   t5[490] := 0.023831;
   t5[491] := 0.0266696;
   t5[492] := 0.0293428;
   t5[493] := 0.0318604;
   t5[494] := 0.0342322;
   t5[495] := -0.0208986;
   t5[496] := -0.0225395;
   t5[497] := -0.0240864;
   t5[498] := -0.0255261;
   t5[499] := -0.0268454;
   t5[500] := -0.0280312;
   t5[501] := -0.0290703;
   t5[502] := -0.0299495;
   t5[503] := -0.0306555;
   t5[504] := -0.0311752;
   t5[505] := -0.0314958;
   t5[506] := -0.0316138;
   t5[507] := -0.0315351;
   t5[508] := -0.0312663;
   t5[509] := -0.0308137;
   t5[510] := -0.0136591;
   t5[511] := -0.0122989;
   t5[512] := -0.0110547;
   t5[513] := -0.0099303;
   t5[514] := -0.0089297;
   t5[515] := -0.0080568;
   t5[516] := -0.0073155;
   t5[517] := -0.0067099;
   t5[518] := -0.0062437;
   t5[519] := -0.0059209;
   t5[520] := -0.0057453;
   t5[521] := -0.0057154;
   t5[522] := -0.0058246;
   t5[523] := -0.006066;
   t5[524] := -0.0064327;
   t5[525] := -0.014299;
   t5[526] := -0.0104196;
   t5[527] := -0.0064601;
   t5[528] := -0.0024202;
   t5[529] := 0.0017005;
   t5[530] := 0.0059023;
   t5[531] := 0.0101856;
   t5[532] := 0.0145506;
   t5[533] := 0.0189979;
   t5[534] := 0.0235277;
   t5[535] := 0.0281401;
   t5[536] := 0.0328307;
   t5[537] := 0.0375902;
   t5[538] := 0.042409;
   t5[539] := 0.0472775;
   t5[540] := -0.0809446;
   t5[541] := -0.0816613;
   t5[542] := -0.0823782;
   t5[543] := -0.0831006;
   t5[544] := -0.0838339;
   t5[545] := -0.0845833;
   t5[546] := -0.0853541;
   t5[547] := -0.0861518;
   t5[548] := -0.0869815;
   t5[549] := -0.0878487;
   t5[550] := -0.0887583;
   t5[551] := -0.0897094;
   t5[552] := -0.0906944;
   t5[553] := -0.0917059;
   t5[554] := -0.092736;
   t5[555] := 0.0001257;
   t5[556] := 0.0029497;
   t5[557] := 0.0057871;
   t5[558] := 0.0086392;
   t5[559] := 0.0115078;
   t5[560] := 0.0143943;
   t5[561] := 0.0173003;
   t5[562] := 0.0202273;
   t5[563] := 0.0231768;
   t5[564] := 0.0261505;
   t5[565] := 0.0291498;
   t5[566] := 0.0321767;
   t5[567] := 0.0352333;
   t5[568] := 0.0383218;
   t5[569] := 0.0414445;
   t5[570] := -0.0673197;
   t5[571] := -0.0670321;
   t5[572] := -0.0666434;
   t5[573] := -0.0661514;
   t5[574] := -0.0655542;
   t5[575] := -0.0648497;
   t5[576] := -0.0640358;
   t5[577] := -0.0631107;
   t5[578] := -0.0620721;
   t5[579] := -0.0609182;
   t5[580] := -0.0596471;
   t5[581] := -0.0582624;
   t5[582] := -0.0567733;
   t5[583] := -0.0551894;
   t5[584] := -0.05352;
   t5[585] := 0.0792828;
   t5[586] := 0.0762561;
   t5[587] := 0.073232;
   t5[588] := 0.0702186;
   t5[589] := 0.067224;
   t5[590] := 0.0642562;
   t5[591] := 0.0613231;
   t5[592] := 0.058433;
   t5[593] := 0.0555937;
   t5[594] := 0.0528132;
   t5[595] := 0.0500996;
   t5[596] := 0.0474569;
   t5[597] := 0.0448857;
   t5[598] := 0.042386;
   t5[599] := 0.0399582;
   t5[600] := -0.1993882;
   t5[601] := -0.1970195;
   t5[602] := -0.1945705;
   t5[603] := -0.1920432;
   t5[604] := -0.1894396;
   t5[605] := -0.1867614;
   t5[606] := -0.1840106;
   t5[607] := -0.1811892;
   t5[608] := -0.1782989;
   t5[609] := -0.1753418;
   t5[610] := -0.1723197;
   t5[611] := -0.1692367;
   t5[612] := -0.1660989;
   t5[613] := -0.1629122;
   t5[614] := -0.159683;
   t5[615] := -0.110986;
   t5[616] := -0.112907;
   t5[617] := -0.1145904;
   t5[618] := -0.11603;
   t5[619] := -0.1172196;
   t5[620] := -0.118153;
   t5[621] := -0.1188239;
   t5[622] := -0.119226;
   t5[623] := -0.1193531;
   t5[624] := -0.1191991;
   t5[625] := -0.1187581;
   t5[626] := -0.1180348;
   t5[627] := -0.1170453;
   t5[628] := -0.1158056;
   t5[629] := -0.1143322;
   t5[630] := -0.0163093;
   t5[631] := -0.0198292;
   t5[632] := -0.0232166;
   t5[633] := -0.0264609;
   t5[634] := -0.0295518;
   t5[635] := -0.0324788;
   t5[636] := -0.0352314;
   t5[637] := -0.0377992;
   t5[638] := -0.0401717;
   t5[639] := -0.0423386;
   t5[640] := -0.0442896;
   t5[641] := -0.0460239;
   t5[642] := -0.0475501;
   t5[643] := -0.0488771;
   t5[644] := -0.0500139;
   t5[645] := 0.0848828;
   t5[646] := 0.0819437;
   t5[647] := 0.0790844;
   t5[648] := 0.0763136;
   t5[649] := 0.0736399;
   t5[650] := 0.0710721;
   t5[651] := 0.0686188;
   t5[652] := 0.0662886;
   t5[653] := 0.0640904;
   t5[654] := 0.0620326;
   t5[655] := 0.0601237;
   t5[656] := 0.0583629;
   t5[657] := 0.05674;
   t5[658] := 0.0552444;
   t5[659] := 0.0538658;
   t5[660] := -0.0819279;
   t5[661] := -0.0837696;
   t5[662] := -0.085415;
   t5[663] := -0.0868444;
   t5[664] := -0.088038;
   t5[665] := -0.0889764;
   t5[666] := -0.0896396;
   t5[667] := -0.0900081;
   t5[668] := -0.0900622;
   t5[669] := -0.0897822;
   t5[670] := -0.0891493;
   t5[671] := -0.0881638;
   t5[672] := -0.0868462;
   t5[673] := -0.0852177;
   t5[674] := -0.0832996;
   t5[675] := -0.0222091;
   t5[676] := -0.019204;
   t5[677] := -0.0163363;
   t5[678] := -0.0136269;
   t5[679] := -0.0110964;
   t5[680] := -0.0087656;
   t5[681] := -0.0066552;
   t5[682] := -0.004786;
   t5[683] := -0.0031786;
   t5[684] := -0.0018538;
   t5[685] := -0.0008317;
   t5[686] := -0.0001178;
   t5[687] := 0.0002977;
   t5[688] := 0.0004254;
   t5[689] := 0.0002755;
   t5[690] := -0.0469918;
   t5[691] := -0.0436484;
   t5[692] := -0.0405246;
   t5[693] := -0.0376308;
   t5[694] := -0.0349775;
   t5[695] := -0.0325752;
   t5[696] := -0.0304344;
   t5[697] := -0.0285657;
   t5[698] := -0.0269795;
   t5[699] := -0.0256863;
   t5[700] := -0.0246962;
   t5[701] := -0.0240066;
   t5[702] := -0.0236022;
   t5[703] := -0.0234672;
   t5[704] := -0.0235855;
   t5[705] := 0.0315658;
   t5[706] := 0.0328791;
   t5[707] := 0.0340612;
   t5[708] := 0.0351116;
   t5[709] := 0.0360298;
   t5[710] := 0.0368152;
   t5[711] := 0.0374672;
   t5[712] := 0.0379854;
   t5[713] := 0.0383692;
   t5[714] := 0.038618;
   t5[715] := 0.0387315;
   t5[716] := 0.0387144;
   t5[717] := 0.0385764;
   t5[718] := 0.0383273;
   t5[719] := 0.0379772;
   t5[720] := 0.0589575;
   t5[721] := 0.0571638;
   t5[722] := 0.0552337;
   t5[723] := 0.0531697;
   t5[724] := 0.0509741;
   t5[725] := 0.0486495;
   t5[726] := 0.0461984;
   t5[727] := 0.0436231;
   t5[728] := 0.0409261;
   t5[729] := 0.03811;
   t5[730] := 0.0351772;
   t5[731] := 0.0321336;
   t5[732] := 0.0289883;
   t5[733] := 0.0257505;
   t5[734] := 0.0224294;
   t5[735] := -0.0370074;
   t5[736] := -0.0344528;
   t5[737] := -0.0317711;
   t5[738] := -0.0289586;
   t5[739] := -0.0260112;
   t5[740] := -0.022925;
   t5[741] := -0.0196963;
   t5[742] := -0.016321;
   t5[743] := -0.0127952;
   t5[744] := -0.0091151;
   t5[745] := -0.005277;
   t5[746] := -0.0012858;
   t5[747] := 0.0028455;
   t5[748] := 0.007103;
   t5[749] := 0.0114734;
   t5[750] := -0.0503424;
   t5[751] := -0.0554995;
   t5[752] := -0.0605443;
   t5[753] := -0.0654624;
   t5[754] := -0.0702395;
   t5[755] := -0.0748614;
   t5[756] := -0.0793139;
   t5[757] := -0.0835825;
   t5[758] := -0.087653;
   t5[759] := -0.0915111;
   t5[760] := -0.095143;
   t5[761] := -0.0985424;
   t5[762] := -0.1017114;
   t5[763] := -0.1046524;
   t5[764] := -0.1073677;
   t5[765] := -0.1648159;
   t5[766] := -0.1596806;
   t5[767] := -0.1543417;
   t5[768] := -0.1488126;
   t5[769] := -0.1431066;
   t5[770] := -0.1372371;
   t5[771] := -0.1312175;
   t5[772] := -0.1250611;
   t5[773] := -0.1187812;
   t5[774] := -0.1123913;
   t5[775] := -0.1059046;
   t5[776] := -0.0993333;
   t5[777] := -0.0926887;
   t5[778] := -0.0859816;
   t5[779] := -0.0792232;
   t5[780] := -0.0904827;
   t5[781] := -0.0898896;
   t5[782] := -0.0893127;
   t5[783] := -0.0887551;
   t5[784] := -0.0882202;
   t5[785] := -0.0877112;
   t5[786] := -0.0872314;
   t5[787] := -0.0867841;
   t5[788] := -0.0863725;
   t5[789] := -0.0859999;
   t5[790] := -0.0856695;
   t5[791] := -0.0853802;
   t5[792] := -0.0851272;
   t5[793] := -0.0849053;
   t5[794] := -0.0847093;
   t5[795] := -0.0673839;
   t5[796] := -0.0627446;
   t5[797] := -0.0580462;
   t5[798] := -0.0533;
   t5[799] := -0.0485171;
   t5[800] := -0.0437086;
   t5[801] := -0.0388857;
   t5[802] := -0.0340594;
   t5[803] := -0.0292411;
   t5[804] := -0.0244417;
   t5[805] := -0.0196723;
   t5[806] := -0.0149416;
   t5[807] := -0.0102555;
   t5[808] := -0.0056201;
   t5[809] := -0.0010412;
   t5[810] := 0.075334;
   t5[811] := 0.0749833;
   t5[812] := 0.0743661;
   t5[813] := 0.0734706;
   t5[814] := 0.072285;
   t5[815] := 0.0707974;
   t5[816] := 0.068996;
   t5[817] := 0.0668689;
   t5[818] := 0.0644045;
   t5[819] := 0.0615908;
   t5[820] := 0.0584166;
   t5[821] := 0.0548866;
   t5[822] := 0.0510212;
   t5[823] := 0.0468419;
   t5[824] := 0.04237;
   t5[825] := -0.1063465;
   t5[826] := -0.1045535;
   t5[827] := -0.1026798;
   t5[828] := -0.1007291;
   t5[829] := -0.0987055;
   t5[830] := -0.0966127;
   t5[831] := -0.0944546;
   t5[832] := -0.092235;
   t5[833] := -0.0899577;
   t5[834] := -0.0876267;
   t5[835] := -0.0852457;
   t5[836] := -0.0828167;
   t5[837] := -0.0803401;
   t5[838] := -0.077816;
   t5[839] := -0.0752449;
   t5[840] := 0.0025241;
   t5[841] := 0.0003729;
   t5[842] := -0.0018117;
   t5[843] := -0.0040243;
   t5[844] := -0.0062591;
   t5[845] := -0.0085107;
   t5[846] := -0.0107734;
   t5[847] := -0.0130416;
   t5[848] := -0.0153097;
   t5[849] := -0.0175722;
   t5[850] := -0.0198235;
   t5[851] := -0.0220606;
   t5[852] := -0.0242824;
   t5[853] := -0.0264882;
   t5[854] := -0.0286772;
   t5[855] := -0.0587365;
   t5[856] := -0.0658987;
   t5[857] := -0.0729648;
   t5[858] := -0.07991;
   t5[859] := -0.0867094;
   t5[860] := -0.0933378;
   t5[861] := -0.0997704;
   t5[862] := -0.1059823;
   t5[863] := -0.1119484;
   t5[864] := -0.1176438;
   t5[865] := -0.1230443;
   t5[866] := -0.1281403;
   t5[867] := -0.1329374;
   t5[868] := -0.137442;
   t5[869] := -0.1416606;
   t5[870] := -0.0241061;
   t5[871] := -0.0227329;
   t5[872] := -0.0212774;
   t5[873] := -0.0197337;
   t5[874] := -0.0180954;
   t5[875] := -0.0163565;
   t5[876] := -0.0145109;
   t5[877] := -0.0125525;
   t5[878] := -0.0104751;
   t5[879] := -0.0082726;
   t5[880] := -0.0059392;
   t5[881] := -0.0034767;
   t5[882] := -0.0008946;
   t5[883] := 0.001797;
   t5[884] := 0.0045883;
   t5[885] := -0.016338;
   t5[886] := -0.0135221;
   t5[887] := -0.0107115;
   t5[888] := -0.0079037;
   t5[889] := -0.0050963;
   t5[890] := -0.0022869;
   t5[891] := 0.0005271;
   t5[892] := 0.0033482;
   t5[893] := 0.0061787;
   t5[894] := 0.0090212;
   t5[895] := 0.011878;
   t5[896] := 0.0147486;
   t5[897] := 0.0176293;
   t5[898] := 0.0205164;
   t5[899] := 0.0234063;
   t5[900] := -0.0519279;
   t5[901] := -0.056473;
   t5[902] := -0.0609004;
   t5[903] := -0.0652012;
   t5[904] := -0.0693667;
   t5[905] := -0.0733882;
   t5[906] := -0.0772569;
   t5[907] := -0.0809641;
   t5[908] := -0.0845011;
   t5[909] := -0.087859;
   t5[910] := -0.0910294;
   t5[911] := -0.0940104;
   t5[912] := -0.0968068;
   t5[913] := -0.0994238;
   t5[914] := -0.1018665;
   t5[915] := 0.142846;
   t5[916] := 0.1405271;
   t5[917] := 0.1380653;
   t5[918] := 0.1354591;
   t5[919] := 0.1327065;
   t5[920] := 0.129806;
   t5[921] := 0.1267559;
   t5[922] := 0.1235543;
   t5[923] := 0.1201996;
   t5[924] := 0.11669;
   t5[925] := 0.1130242;
   t5[926] := 0.109206;
   t5[927] := 0.1052453;
   t5[928] := 0.1011521;
   t5[929] := 0.0969364;
   t5[930] := -0.0299947;
   t5[931] := -0.0294521;
   t5[932] := -0.0288785;
   t5[933] := -0.0282723;
   t5[934] := -0.0276319;
   t5[935] := -0.0269553;
   t5[936] := -0.0262411;
   t5[937] := -0.0254874;
   t5[938] := -0.0246926;
   t5[939] := -0.0238549;
   t5[940] := -0.0229728;
   t5[941] := -0.0220476;
   t5[942] := -0.0210837;
   t5[943] := -0.0200855;
   t5[944] := -0.0190576;
   t5[945] := -0.0100999;
   t5[946] := -0.0030712;
   t5[947] := 0.0037406;
   t5[948] := 0.0103103;
   t5[949] := 0.0166126;
   t5[950] := 0.0226221;
   t5[951] := 0.0283136;
   t5[952] := 0.0336617;
   t5[953] := 0.038641;
   t5[954] := 0.0432264;
   t5[955] := 0.0473932;
   t5[956] := 0.0511381;
   t5[957] := 0.054479;
   t5[958] := 0.0574348;
   t5[959] := 0.0600244;
   w6[0] := 0.0254122;
   w6[1] := -0.4251655;
   w6[2] := -0.4513899;
   w6[3] := 0.0262705;
   w6[4] := 0.3702881;
   w6[5] := -0.1208161;
   w6[6] := -0.2231239;
   w6[7] := 0.2512441;
   w6[8] := -0.3278799;
   w6[9] := 0.2889541;
   w6[10] := -0.0654242;
   w6[11] := 0.1067281;
   w6[12] := 0.2623815;
   w6[13] := -0.1798091;
   w6[14] := -0.3070911;
   w6[15] := -0.4204447;
   w6[16] := 0.5762351;
   w6[17] := -1.090657;
   w6[18] := -0.2690518;
   w6[19] := -0.6730261;
   w6[20] := -0.0514923;
   w6[21] := -0.4457789;
   w6[22] := 0.5072183;
   w6[23] := -0.0549661;
   w6[24] := 0.3812394;
   w6[25] := -0.606307;
   w6[26] := 0.1917919;
   w6[27] := 0.1525442;
   w6[28] := -0.4219312;
   w6[29] := 0.338313;
   w6[30] := 0.1919874;
   w6[31] := -0.3457294;
   w6[32] := 0.1728978;
   w6[33] := 0.5825878;
   w6[34] := 0.7331663;
   w6[35] := 0.4268312;
   w6[36] := -0.0077422;
   w6[37] := 0.4766487;
   w6[38] := 0.102607;
   w6[39] := -0.5723706;
   w6[40] := 0.0728498;
   w6[41] := 0.4253429;
   w6[42] := -0.3637053;
   w6[43] := -0.6206156;
   w6[44] := 0.2656944;
   w6[45] := -0.3130539;
   w6[46] := 0.2033212;
   w6[47] := 0.1327122;
   w6[48] := -0.709101;
   w6[49] := 0.7231103;
   w6[50] := -0.2214241;
   w6[51] := 0.4491622;
   w6[52] := -0.3655713;
   w6[53] := 0.4263724;
   w6[54] := 0.0266531;
   w6[55] := 0.4637966;
   w6[56] := -0.3418979;
   w6[57] := -0.2391363;
   w6[58] := 0.4152579;
   w6[59] := 0.2146362;
   w6[60] := -0.3901598;
   w6[61] := -0.1938754;
   w6[62] := -0.561949;
   w6[63] := 0.4047181;
END_DATA_BLOCK

FUNCTION_BLOCK "NeuroPLC_Inference"   // FB1, SCL
{ S7_Optimized_Access := 'FALSE' }
VERSION : 0.1
// NeuroPLC 鈥?Auto-generated IEC 61131-3 SCL (DB+FB Mode)
//  Graph: kan | Target: S71200DBBackend
//  Work memory: 75KB | LUT points: 15
//  Nodes: 11 | Ops: {'matmul': 3, 'standard_act': 2, 'bspline_lut': 2, 'add': 2, 'softmax': 1, 'argmax': 1}
//  Parameters in DB "NeuroPLC_KAN_Weights", inference in FB.
   VAR_INPUT
      features : Array[0..27] of Real;   // 28-D feature vector
   END_VAR
   VAR_OUTPUT
      fault_class : Int;   // 0=Normal, 1=InnerRace, 2=Ball, 3=OuterRace
      confidence : Real;   // max softmax probability 鈹€鈹€ Inference temporaries 鈹€鈹€
   END_VAR
   VAR
      v1 : Array[0..27] of Real;   // silu output
      v3 : Array[0..447] of Real;   // BsplineLUT output (1D: o*28+i)
      v2 : Array[0..15] of Real;   // matmul output
      v4 : Array[0..15] of Real;   // add merge
      v5 : Array[0..15] of Real;   // silu output
      v7 : Array[0..63] of Real;   // BsplineLUT output (1D: o*16+i)
      v6 : Array[0..3] of Real;   // matmul output
      v8 : Array[0..3] of Real;   // add merge
      v9 : Array[0..3] of Real;   // softmax output 鈹€鈹€ Temporary variables 鈹€鈹€
      i : Int;
      o : Int;
      j : Int;
      lo : Int;
      hi : Int;
      idx : Int;
      base : Int;
      sum : Real;
      max_val : Real;
      t_val : Real;
   END_VAR
BEGIN
      // 鈺愨晲鈺?Inference forward pass 鈺愨晲鈺?
       // Parameters loaded from DB "NeuroPLC_KAN_Weights" (start values = data, not code)

          // Input: features[0..27]

          // StandardAct: silu
          FOR #i := 0 TO 27 DO
              // SiLU = x / (1 + exp(-x))
              #v1[#i] := #features[#i] / (1.0 + EXP(-#features[#i]));
          END_FOR;

          // BsplineLUT: l0_bspline (16x28, 15 pts)
          FOR #i := 0 TO 27 DO
              // Linear scan: find largest grid[j] <= input[i]
              #lo := 0;
              FOR #j := 1 TO 13 DO
                  IF #features[#i] >= "NeuroPLC_KAN_Weights".g0[#j] THEN
                      #lo := #j;
                  END_IF;
              END_FOR;
              #hi := #lo + 1;
              #t_val := (#features[#i] - "NeuroPLC_KAN_Weights".g0[#lo]) /
                        ("NeuroPLC_KAN_Weights".g0[#hi] - "NeuroPLC_KAN_Weights".g0[#lo] + 1.0E-10);
              FOR #o := 0 TO 15 DO
                  #base := (#o * 28 + #i) * 15;
                  #idx := #o * 28 + #i;
                  #v3[#idx] :=
                      "NeuroPLC_KAN_Weights".t1[#base + #lo] * (1.0 - #t_val) +
                      "NeuroPLC_KAN_Weights".t1[#base + #hi] * #t_val;
              END_FOR;
          END_FOR;

          // MatMul: l0_base
          #v2[0] := "NeuroPLC_KAN_Weights".b3[0] + "NeuroPLC_KAN_Weights".w2[0] * #v1[0] + "NeuroPLC_KAN_Weights".w2[1] * #v1[1] + "NeuroPLC_KAN_Weights".w2[2] * #v1[2] + "NeuroPLC_KAN_Weights".w2[3] * #v1[3] + "NeuroPLC_KAN_Weights".w2[4] * #v1[4] + "NeuroPLC_KAN_Weights".w2[5] * #v1[5] + "NeuroPLC_KAN_Weights".w2[6] * #v1[6] + "NeuroPLC_KAN_Weights".w2[7] * #v1[7] + "NeuroPLC_KAN_Weights".w2[8] * #v1[8] + "NeuroPLC_KAN_Weights".w2[9] * #v1[9] + "NeuroPLC_KAN_Weights".w2[10] * #v1[10] + "NeuroPLC_KAN_Weights".w2[11] * #v1[11] + "NeuroPLC_KAN_Weights".w2[12] * #v1[12] + "NeuroPLC_KAN_Weights".w2[13] * #v1[13] + "NeuroPLC_KAN_Weights".w2[14] * #v1[14] + "NeuroPLC_KAN_Weights".w2[15] * #v1[15] + "NeuroPLC_KAN_Weights".w2[16] * #v1[16] + "NeuroPLC_KAN_Weights".w2[17] * #v1[17] + "NeuroPLC_KAN_Weights".w2[18] * #v1[18] + "NeuroPLC_KAN_Weights".w2[19] * #v1[19] + "NeuroPLC_KAN_Weights".w2[20] * #v1[20] + "NeuroPLC_KAN_Weights".w2[21] * #v1[21] + "NeuroPLC_KAN_Weights".w2[22] * #v1[22] + "NeuroPLC_KAN_Weights".w2[23] * #v1[23] + "NeuroPLC_KAN_Weights".w2[24] * #v1[24] + "NeuroPLC_KAN_Weights".w2[25] * #v1[25] + "NeuroPLC_KAN_Weights".w2[26] * #v1[26] + "NeuroPLC_KAN_Weights".w2[27] * #v1[27];
          #v2[1] := "NeuroPLC_KAN_Weights".b3[1] + "NeuroPLC_KAN_Weights".w2[28] * #v1[0] + "NeuroPLC_KAN_Weights".w2[29] * #v1[1] + "NeuroPLC_KAN_Weights".w2[30] * #v1[2] + "NeuroPLC_KAN_Weights".w2[31] * #v1[3] + "NeuroPLC_KAN_Weights".w2[32] * #v1[4] + "NeuroPLC_KAN_Weights".w2[33] * #v1[5] + "NeuroPLC_KAN_Weights".w2[34] * #v1[6] + "NeuroPLC_KAN_Weights".w2[35] * #v1[7] + "NeuroPLC_KAN_Weights".w2[36] * #v1[8] + "NeuroPLC_KAN_Weights".w2[37] * #v1[9] + "NeuroPLC_KAN_Weights".w2[38] * #v1[10] + "NeuroPLC_KAN_Weights".w2[39] * #v1[11] + "NeuroPLC_KAN_Weights".w2[40] * #v1[12] + "NeuroPLC_KAN_Weights".w2[41] * #v1[13] + "NeuroPLC_KAN_Weights".w2[42] * #v1[14] + "NeuroPLC_KAN_Weights".w2[43] * #v1[15] + "NeuroPLC_KAN_Weights".w2[44] * #v1[16] + "NeuroPLC_KAN_Weights".w2[45] * #v1[17] + "NeuroPLC_KAN_Weights".w2[46] * #v1[18] + "NeuroPLC_KAN_Weights".w2[47] * #v1[19] + "NeuroPLC_KAN_Weights".w2[48] * #v1[20] + "NeuroPLC_KAN_Weights".w2[49] * #v1[21] + "NeuroPLC_KAN_Weights".w2[50] * #v1[22] + "NeuroPLC_KAN_Weights".w2[51] * #v1[23] + "NeuroPLC_KAN_Weights".w2[52] * #v1[24] + "NeuroPLC_KAN_Weights".w2[53] * #v1[25] + "NeuroPLC_KAN_Weights".w2[54] * #v1[26] + "NeuroPLC_KAN_Weights".w2[55] * #v1[27];
          #v2[2] := "NeuroPLC_KAN_Weights".b3[2] + "NeuroPLC_KAN_Weights".w2[56] * #v1[0] + "NeuroPLC_KAN_Weights".w2[57] * #v1[1] + "NeuroPLC_KAN_Weights".w2[58] * #v1[2] + "NeuroPLC_KAN_Weights".w2[59] * #v1[3] + "NeuroPLC_KAN_Weights".w2[60] * #v1[4] + "NeuroPLC_KAN_Weights".w2[61] * #v1[5] + "NeuroPLC_KAN_Weights".w2[62] * #v1[6] + "NeuroPLC_KAN_Weights".w2[63] * #v1[7] + "NeuroPLC_KAN_Weights".w2[64] * #v1[8] + "NeuroPLC_KAN_Weights".w2[65] * #v1[9] + "NeuroPLC_KAN_Weights".w2[66] * #v1[10] + "NeuroPLC_KAN_Weights".w2[67] * #v1[11] + "NeuroPLC_KAN_Weights".w2[68] * #v1[12] + "NeuroPLC_KAN_Weights".w2[69] * #v1[13] + "NeuroPLC_KAN_Weights".w2[70] * #v1[14] + "NeuroPLC_KAN_Weights".w2[71] * #v1[15] + "NeuroPLC_KAN_Weights".w2[72] * #v1[16] + "NeuroPLC_KAN_Weights".w2[73] * #v1[17] + "NeuroPLC_KAN_Weights".w2[74] * #v1[18] + "NeuroPLC_KAN_Weights".w2[75] * #v1[19] + "NeuroPLC_KAN_Weights".w2[76] * #v1[20] + "NeuroPLC_KAN_Weights".w2[77] * #v1[21] + "NeuroPLC_KAN_Weights".w2[78] * #v1[22] + "NeuroPLC_KAN_Weights".w2[79] * #v1[23] + "NeuroPLC_KAN_Weights".w2[80] * #v1[24] + "NeuroPLC_KAN_Weights".w2[81] * #v1[25] + "NeuroPLC_KAN_Weights".w2[82] * #v1[26] + "NeuroPLC_KAN_Weights".w2[83] * #v1[27];
          #v2[3] := "NeuroPLC_KAN_Weights".b3[3] + "NeuroPLC_KAN_Weights".w2[84] * #v1[0] + "NeuroPLC_KAN_Weights".w2[85] * #v1[1] + "NeuroPLC_KAN_Weights".w2[86] * #v1[2] + "NeuroPLC_KAN_Weights".w2[87] * #v1[3] + "NeuroPLC_KAN_Weights".w2[88] * #v1[4] + "NeuroPLC_KAN_Weights".w2[89] * #v1[5] + "NeuroPLC_KAN_Weights".w2[90] * #v1[6] + "NeuroPLC_KAN_Weights".w2[91] * #v1[7] + "NeuroPLC_KAN_Weights".w2[92] * #v1[8] + "NeuroPLC_KAN_Weights".w2[93] * #v1[9] + "NeuroPLC_KAN_Weights".w2[94] * #v1[10] + "NeuroPLC_KAN_Weights".w2[95] * #v1[11] + "NeuroPLC_KAN_Weights".w2[96] * #v1[12] + "NeuroPLC_KAN_Weights".w2[97] * #v1[13] + "NeuroPLC_KAN_Weights".w2[98] * #v1[14] + "NeuroPLC_KAN_Weights".w2[99] * #v1[15] + "NeuroPLC_KAN_Weights".w2[100] * #v1[16] + "NeuroPLC_KAN_Weights".w2[101] * #v1[17] + "NeuroPLC_KAN_Weights".w2[102] * #v1[18] + "NeuroPLC_KAN_Weights".w2[103] * #v1[19] + "NeuroPLC_KAN_Weights".w2[104] * #v1[20] + "NeuroPLC_KAN_Weights".w2[105] * #v1[21] + "NeuroPLC_KAN_Weights".w2[106] * #v1[22] + "NeuroPLC_KAN_Weights".w2[107] * #v1[23] + "NeuroPLC_KAN_Weights".w2[108] * #v1[24] + "NeuroPLC_KAN_Weights".w2[109] * #v1[25] + "NeuroPLC_KAN_Weights".w2[110] * #v1[26] + "NeuroPLC_KAN_Weights".w2[111] * #v1[27];
          #v2[4] := "NeuroPLC_KAN_Weights".b3[4] + "NeuroPLC_KAN_Weights".w2[112] * #v1[0] + "NeuroPLC_KAN_Weights".w2[113] * #v1[1] + "NeuroPLC_KAN_Weights".w2[114] * #v1[2] + "NeuroPLC_KAN_Weights".w2[115] * #v1[3] + "NeuroPLC_KAN_Weights".w2[116] * #v1[4] + "NeuroPLC_KAN_Weights".w2[117] * #v1[5] + "NeuroPLC_KAN_Weights".w2[118] * #v1[6] + "NeuroPLC_KAN_Weights".w2[119] * #v1[7] + "NeuroPLC_KAN_Weights".w2[120] * #v1[8] + "NeuroPLC_KAN_Weights".w2[121] * #v1[9] + "NeuroPLC_KAN_Weights".w2[122] * #v1[10] + "NeuroPLC_KAN_Weights".w2[123] * #v1[11] + "NeuroPLC_KAN_Weights".w2[124] * #v1[12] + "NeuroPLC_KAN_Weights".w2[125] * #v1[13] + "NeuroPLC_KAN_Weights".w2[126] * #v1[14] + "NeuroPLC_KAN_Weights".w2[127] * #v1[15] + "NeuroPLC_KAN_Weights".w2[128] * #v1[16] + "NeuroPLC_KAN_Weights".w2[129] * #v1[17] + "NeuroPLC_KAN_Weights".w2[130] * #v1[18] + "NeuroPLC_KAN_Weights".w2[131] * #v1[19] + "NeuroPLC_KAN_Weights".w2[132] * #v1[20] + "NeuroPLC_KAN_Weights".w2[133] * #v1[21] + "NeuroPLC_KAN_Weights".w2[134] * #v1[22] + "NeuroPLC_KAN_Weights".w2[135] * #v1[23] + "NeuroPLC_KAN_Weights".w2[136] * #v1[24] + "NeuroPLC_KAN_Weights".w2[137] * #v1[25] + "NeuroPLC_KAN_Weights".w2[138] * #v1[26] + "NeuroPLC_KAN_Weights".w2[139] * #v1[27];
          #v2[5] := "NeuroPLC_KAN_Weights".b3[5] + "NeuroPLC_KAN_Weights".w2[140] * #v1[0] + "NeuroPLC_KAN_Weights".w2[141] * #v1[1] + "NeuroPLC_KAN_Weights".w2[142] * #v1[2] + "NeuroPLC_KAN_Weights".w2[143] * #v1[3] + "NeuroPLC_KAN_Weights".w2[144] * #v1[4] + "NeuroPLC_KAN_Weights".w2[145] * #v1[5] + "NeuroPLC_KAN_Weights".w2[146] * #v1[6] + "NeuroPLC_KAN_Weights".w2[147] * #v1[7] + "NeuroPLC_KAN_Weights".w2[148] * #v1[8] + "NeuroPLC_KAN_Weights".w2[149] * #v1[9] + "NeuroPLC_KAN_Weights".w2[150] * #v1[10] + "NeuroPLC_KAN_Weights".w2[151] * #v1[11] + "NeuroPLC_KAN_Weights".w2[152] * #v1[12] + "NeuroPLC_KAN_Weights".w2[153] * #v1[13] + "NeuroPLC_KAN_Weights".w2[154] * #v1[14] + "NeuroPLC_KAN_Weights".w2[155] * #v1[15] + "NeuroPLC_KAN_Weights".w2[156] * #v1[16] + "NeuroPLC_KAN_Weights".w2[157] * #v1[17] + "NeuroPLC_KAN_Weights".w2[158] * #v1[18] + "NeuroPLC_KAN_Weights".w2[159] * #v1[19] + "NeuroPLC_KAN_Weights".w2[160] * #v1[20] + "NeuroPLC_KAN_Weights".w2[161] * #v1[21] + "NeuroPLC_KAN_Weights".w2[162] * #v1[22] + "NeuroPLC_KAN_Weights".w2[163] * #v1[23] + "NeuroPLC_KAN_Weights".w2[164] * #v1[24] + "NeuroPLC_KAN_Weights".w2[165] * #v1[25] + "NeuroPLC_KAN_Weights".w2[166] * #v1[26] + "NeuroPLC_KAN_Weights".w2[167] * #v1[27];
          #v2[6] := "NeuroPLC_KAN_Weights".b3[6] + "NeuroPLC_KAN_Weights".w2[168] * #v1[0] + "NeuroPLC_KAN_Weights".w2[169] * #v1[1] + "NeuroPLC_KAN_Weights".w2[170] * #v1[2] + "NeuroPLC_KAN_Weights".w2[171] * #v1[3] + "NeuroPLC_KAN_Weights".w2[172] * #v1[4] + "NeuroPLC_KAN_Weights".w2[173] * #v1[5] + "NeuroPLC_KAN_Weights".w2[174] * #v1[6] + "NeuroPLC_KAN_Weights".w2[175] * #v1[7] + "NeuroPLC_KAN_Weights".w2[176] * #v1[8] + "NeuroPLC_KAN_Weights".w2[177] * #v1[9] + "NeuroPLC_KAN_Weights".w2[178] * #v1[10] + "NeuroPLC_KAN_Weights".w2[179] * #v1[11] + "NeuroPLC_KAN_Weights".w2[180] * #v1[12] + "NeuroPLC_KAN_Weights".w2[181] * #v1[13] + "NeuroPLC_KAN_Weights".w2[182] * #v1[14] + "NeuroPLC_KAN_Weights".w2[183] * #v1[15] + "NeuroPLC_KAN_Weights".w2[184] * #v1[16] + "NeuroPLC_KAN_Weights".w2[185] * #v1[17] + "NeuroPLC_KAN_Weights".w2[186] * #v1[18] + "NeuroPLC_KAN_Weights".w2[187] * #v1[19] + "NeuroPLC_KAN_Weights".w2[188] * #v1[20] + "NeuroPLC_KAN_Weights".w2[189] * #v1[21] + "NeuroPLC_KAN_Weights".w2[190] * #v1[22] + "NeuroPLC_KAN_Weights".w2[191] * #v1[23] + "NeuroPLC_KAN_Weights".w2[192] * #v1[24] + "NeuroPLC_KAN_Weights".w2[193] * #v1[25] + "NeuroPLC_KAN_Weights".w2[194] * #v1[26] + "NeuroPLC_KAN_Weights".w2[195] * #v1[27];
          #v2[7] := "NeuroPLC_KAN_Weights".b3[7] + "NeuroPLC_KAN_Weights".w2[196] * #v1[0] + "NeuroPLC_KAN_Weights".w2[197] * #v1[1] + "NeuroPLC_KAN_Weights".w2[198] * #v1[2] + "NeuroPLC_KAN_Weights".w2[199] * #v1[3] + "NeuroPLC_KAN_Weights".w2[200] * #v1[4] + "NeuroPLC_KAN_Weights".w2[201] * #v1[5] + "NeuroPLC_KAN_Weights".w2[202] * #v1[6] + "NeuroPLC_KAN_Weights".w2[203] * #v1[7] + "NeuroPLC_KAN_Weights".w2[204] * #v1[8] + "NeuroPLC_KAN_Weights".w2[205] * #v1[9] + "NeuroPLC_KAN_Weights".w2[206] * #v1[10] + "NeuroPLC_KAN_Weights".w2[207] * #v1[11] + "NeuroPLC_KAN_Weights".w2[208] * #v1[12] + "NeuroPLC_KAN_Weights".w2[209] * #v1[13] + "NeuroPLC_KAN_Weights".w2[210] * #v1[14] + "NeuroPLC_KAN_Weights".w2[211] * #v1[15] + "NeuroPLC_KAN_Weights".w2[212] * #v1[16] + "NeuroPLC_KAN_Weights".w2[213] * #v1[17] + "NeuroPLC_KAN_Weights".w2[214] * #v1[18] + "NeuroPLC_KAN_Weights".w2[215] * #v1[19] + "NeuroPLC_KAN_Weights".w2[216] * #v1[20] + "NeuroPLC_KAN_Weights".w2[217] * #v1[21] + "NeuroPLC_KAN_Weights".w2[218] * #v1[22] + "NeuroPLC_KAN_Weights".w2[219] * #v1[23] + "NeuroPLC_KAN_Weights".w2[220] * #v1[24] + "NeuroPLC_KAN_Weights".w2[221] * #v1[25] + "NeuroPLC_KAN_Weights".w2[222] * #v1[26] + "NeuroPLC_KAN_Weights".w2[223] * #v1[27];
          #v2[8] := "NeuroPLC_KAN_Weights".b3[8] + "NeuroPLC_KAN_Weights".w2[224] * #v1[0] + "NeuroPLC_KAN_Weights".w2[225] * #v1[1] + "NeuroPLC_KAN_Weights".w2[226] * #v1[2] + "NeuroPLC_KAN_Weights".w2[227] * #v1[3] + "NeuroPLC_KAN_Weights".w2[228] * #v1[4] + "NeuroPLC_KAN_Weights".w2[229] * #v1[5] + "NeuroPLC_KAN_Weights".w2[230] * #v1[6] + "NeuroPLC_KAN_Weights".w2[231] * #v1[7] + "NeuroPLC_KAN_Weights".w2[232] * #v1[8] + "NeuroPLC_KAN_Weights".w2[233] * #v1[9] + "NeuroPLC_KAN_Weights".w2[234] * #v1[10] + "NeuroPLC_KAN_Weights".w2[235] * #v1[11] + "NeuroPLC_KAN_Weights".w2[236] * #v1[12] + "NeuroPLC_KAN_Weights".w2[237] * #v1[13] + "NeuroPLC_KAN_Weights".w2[238] * #v1[14] + "NeuroPLC_KAN_Weights".w2[239] * #v1[15] + "NeuroPLC_KAN_Weights".w2[240] * #v1[16] + "NeuroPLC_KAN_Weights".w2[241] * #v1[17] + "NeuroPLC_KAN_Weights".w2[242] * #v1[18] + "NeuroPLC_KAN_Weights".w2[243] * #v1[19] + "NeuroPLC_KAN_Weights".w2[244] * #v1[20] + "NeuroPLC_KAN_Weights".w2[245] * #v1[21] + "NeuroPLC_KAN_Weights".w2[246] * #v1[22] + "NeuroPLC_KAN_Weights".w2[247] * #v1[23] + "NeuroPLC_KAN_Weights".w2[248] * #v1[24] + "NeuroPLC_KAN_Weights".w2[249] * #v1[25] + "NeuroPLC_KAN_Weights".w2[250] * #v1[26] + "NeuroPLC_KAN_Weights".w2[251] * #v1[27];
          #v2[9] := "NeuroPLC_KAN_Weights".b3[9] + "NeuroPLC_KAN_Weights".w2[252] * #v1[0] + "NeuroPLC_KAN_Weights".w2[253] * #v1[1] + "NeuroPLC_KAN_Weights".w2[254] * #v1[2] + "NeuroPLC_KAN_Weights".w2[255] * #v1[3] + "NeuroPLC_KAN_Weights".w2[256] * #v1[4] + "NeuroPLC_KAN_Weights".w2[257] * #v1[5] + "NeuroPLC_KAN_Weights".w2[258] * #v1[6] + "NeuroPLC_KAN_Weights".w2[259] * #v1[7] + "NeuroPLC_KAN_Weights".w2[260] * #v1[8] + "NeuroPLC_KAN_Weights".w2[261] * #v1[9] + "NeuroPLC_KAN_Weights".w2[262] * #v1[10] + "NeuroPLC_KAN_Weights".w2[263] * #v1[11] + "NeuroPLC_KAN_Weights".w2[264] * #v1[12] + "NeuroPLC_KAN_Weights".w2[265] * #v1[13] + "NeuroPLC_KAN_Weights".w2[266] * #v1[14] + "NeuroPLC_KAN_Weights".w2[267] * #v1[15] + "NeuroPLC_KAN_Weights".w2[268] * #v1[16] + "NeuroPLC_KAN_Weights".w2[269] * #v1[17] + "NeuroPLC_KAN_Weights".w2[270] * #v1[18] + "NeuroPLC_KAN_Weights".w2[271] * #v1[19] + "NeuroPLC_KAN_Weights".w2[272] * #v1[20] + "NeuroPLC_KAN_Weights".w2[273] * #v1[21] + "NeuroPLC_KAN_Weights".w2[274] * #v1[22] + "NeuroPLC_KAN_Weights".w2[275] * #v1[23] + "NeuroPLC_KAN_Weights".w2[276] * #v1[24] + "NeuroPLC_KAN_Weights".w2[277] * #v1[25] + "NeuroPLC_KAN_Weights".w2[278] * #v1[26] + "NeuroPLC_KAN_Weights".w2[279] * #v1[27];
          #v2[10] := "NeuroPLC_KAN_Weights".b3[10] + "NeuroPLC_KAN_Weights".w2[280] * #v1[0] + "NeuroPLC_KAN_Weights".w2[281] * #v1[1] + "NeuroPLC_KAN_Weights".w2[282] * #v1[2] + "NeuroPLC_KAN_Weights".w2[283] * #v1[3] + "NeuroPLC_KAN_Weights".w2[284] * #v1[4] + "NeuroPLC_KAN_Weights".w2[285] * #v1[5] + "NeuroPLC_KAN_Weights".w2[286] * #v1[6] + "NeuroPLC_KAN_Weights".w2[287] * #v1[7] + "NeuroPLC_KAN_Weights".w2[288] * #v1[8] + "NeuroPLC_KAN_Weights".w2[289] * #v1[9] + "NeuroPLC_KAN_Weights".w2[290] * #v1[10] + "NeuroPLC_KAN_Weights".w2[291] * #v1[11] + "NeuroPLC_KAN_Weights".w2[292] * #v1[12] + "NeuroPLC_KAN_Weights".w2[293] * #v1[13] + "NeuroPLC_KAN_Weights".w2[294] * #v1[14] + "NeuroPLC_KAN_Weights".w2[295] * #v1[15] + "NeuroPLC_KAN_Weights".w2[296] * #v1[16] + "NeuroPLC_KAN_Weights".w2[297] * #v1[17] + "NeuroPLC_KAN_Weights".w2[298] * #v1[18] + "NeuroPLC_KAN_Weights".w2[299] * #v1[19] + "NeuroPLC_KAN_Weights".w2[300] * #v1[20] + "NeuroPLC_KAN_Weights".w2[301] * #v1[21] + "NeuroPLC_KAN_Weights".w2[302] * #v1[22] + "NeuroPLC_KAN_Weights".w2[303] * #v1[23] + "NeuroPLC_KAN_Weights".w2[304] * #v1[24] + "NeuroPLC_KAN_Weights".w2[305] * #v1[25] + "NeuroPLC_KAN_Weights".w2[306] * #v1[26] + "NeuroPLC_KAN_Weights".w2[307] * #v1[27];
          #v2[11] := "NeuroPLC_KAN_Weights".b3[11] + "NeuroPLC_KAN_Weights".w2[308] * #v1[0] + "NeuroPLC_KAN_Weights".w2[309] * #v1[1] + "NeuroPLC_KAN_Weights".w2[310] * #v1[2] + "NeuroPLC_KAN_Weights".w2[311] * #v1[3] + "NeuroPLC_KAN_Weights".w2[312] * #v1[4] + "NeuroPLC_KAN_Weights".w2[313] * #v1[5] + "NeuroPLC_KAN_Weights".w2[314] * #v1[6] + "NeuroPLC_KAN_Weights".w2[315] * #v1[7] + "NeuroPLC_KAN_Weights".w2[316] * #v1[8] + "NeuroPLC_KAN_Weights".w2[317] * #v1[9] + "NeuroPLC_KAN_Weights".w2[318] * #v1[10] + "NeuroPLC_KAN_Weights".w2[319] * #v1[11] + "NeuroPLC_KAN_Weights".w2[320] * #v1[12] + "NeuroPLC_KAN_Weights".w2[321] * #v1[13] + "NeuroPLC_KAN_Weights".w2[322] * #v1[14] + "NeuroPLC_KAN_Weights".w2[323] * #v1[15] + "NeuroPLC_KAN_Weights".w2[324] * #v1[16] + "NeuroPLC_KAN_Weights".w2[325] * #v1[17] + "NeuroPLC_KAN_Weights".w2[326] * #v1[18] + "NeuroPLC_KAN_Weights".w2[327] * #v1[19] + "NeuroPLC_KAN_Weights".w2[328] * #v1[20] + "NeuroPLC_KAN_Weights".w2[329] * #v1[21] + "NeuroPLC_KAN_Weights".w2[330] * #v1[22] + "NeuroPLC_KAN_Weights".w2[331] * #v1[23] + "NeuroPLC_KAN_Weights".w2[332] * #v1[24] + "NeuroPLC_KAN_Weights".w2[333] * #v1[25] + "NeuroPLC_KAN_Weights".w2[334] * #v1[26] + "NeuroPLC_KAN_Weights".w2[335] * #v1[27];
          #v2[12] := "NeuroPLC_KAN_Weights".b3[12] + "NeuroPLC_KAN_Weights".w2[336] * #v1[0] + "NeuroPLC_KAN_Weights".w2[337] * #v1[1] + "NeuroPLC_KAN_Weights".w2[338] * #v1[2] + "NeuroPLC_KAN_Weights".w2[339] * #v1[3] + "NeuroPLC_KAN_Weights".w2[340] * #v1[4] + "NeuroPLC_KAN_Weights".w2[341] * #v1[5] + "NeuroPLC_KAN_Weights".w2[342] * #v1[6] + "NeuroPLC_KAN_Weights".w2[343] * #v1[7] + "NeuroPLC_KAN_Weights".w2[344] * #v1[8] + "NeuroPLC_KAN_Weights".w2[345] * #v1[9] + "NeuroPLC_KAN_Weights".w2[346] * #v1[10] + "NeuroPLC_KAN_Weights".w2[347] * #v1[11] + "NeuroPLC_KAN_Weights".w2[348] * #v1[12] + "NeuroPLC_KAN_Weights".w2[349] * #v1[13] + "NeuroPLC_KAN_Weights".w2[350] * #v1[14] + "NeuroPLC_KAN_Weights".w2[351] * #v1[15] + "NeuroPLC_KAN_Weights".w2[352] * #v1[16] + "NeuroPLC_KAN_Weights".w2[353] * #v1[17] + "NeuroPLC_KAN_Weights".w2[354] * #v1[18] + "NeuroPLC_KAN_Weights".w2[355] * #v1[19] + "NeuroPLC_KAN_Weights".w2[356] * #v1[20] + "NeuroPLC_KAN_Weights".w2[357] * #v1[21] + "NeuroPLC_KAN_Weights".w2[358] * #v1[22] + "NeuroPLC_KAN_Weights".w2[359] * #v1[23] + "NeuroPLC_KAN_Weights".w2[360] * #v1[24] + "NeuroPLC_KAN_Weights".w2[361] * #v1[25] + "NeuroPLC_KAN_Weights".w2[362] * #v1[26] + "NeuroPLC_KAN_Weights".w2[363] * #v1[27];
          #v2[13] := "NeuroPLC_KAN_Weights".b3[13] + "NeuroPLC_KAN_Weights".w2[364] * #v1[0] + "NeuroPLC_KAN_Weights".w2[365] * #v1[1] + "NeuroPLC_KAN_Weights".w2[366] * #v1[2] + "NeuroPLC_KAN_Weights".w2[367] * #v1[3] + "NeuroPLC_KAN_Weights".w2[368] * #v1[4] + "NeuroPLC_KAN_Weights".w2[369] * #v1[5] + "NeuroPLC_KAN_Weights".w2[370] * #v1[6] + "NeuroPLC_KAN_Weights".w2[371] * #v1[7] + "NeuroPLC_KAN_Weights".w2[372] * #v1[8] + "NeuroPLC_KAN_Weights".w2[373] * #v1[9] + "NeuroPLC_KAN_Weights".w2[374] * #v1[10] + "NeuroPLC_KAN_Weights".w2[375] * #v1[11] + "NeuroPLC_KAN_Weights".w2[376] * #v1[12] + "NeuroPLC_KAN_Weights".w2[377] * #v1[13] + "NeuroPLC_KAN_Weights".w2[378] * #v1[14] + "NeuroPLC_KAN_Weights".w2[379] * #v1[15] + "NeuroPLC_KAN_Weights".w2[380] * #v1[16] + "NeuroPLC_KAN_Weights".w2[381] * #v1[17] + "NeuroPLC_KAN_Weights".w2[382] * #v1[18] + "NeuroPLC_KAN_Weights".w2[383] * #v1[19] + "NeuroPLC_KAN_Weights".w2[384] * #v1[20] + "NeuroPLC_KAN_Weights".w2[385] * #v1[21] + "NeuroPLC_KAN_Weights".w2[386] * #v1[22] + "NeuroPLC_KAN_Weights".w2[387] * #v1[23] + "NeuroPLC_KAN_Weights".w2[388] * #v1[24] + "NeuroPLC_KAN_Weights".w2[389] * #v1[25] + "NeuroPLC_KAN_Weights".w2[390] * #v1[26] + "NeuroPLC_KAN_Weights".w2[391] * #v1[27];
          #v2[14] := "NeuroPLC_KAN_Weights".b3[14] + "NeuroPLC_KAN_Weights".w2[392] * #v1[0] + "NeuroPLC_KAN_Weights".w2[393] * #v1[1] + "NeuroPLC_KAN_Weights".w2[394] * #v1[2] + "NeuroPLC_KAN_Weights".w2[395] * #v1[3] + "NeuroPLC_KAN_Weights".w2[396] * #v1[4] + "NeuroPLC_KAN_Weights".w2[397] * #v1[5] + "NeuroPLC_KAN_Weights".w2[398] * #v1[6] + "NeuroPLC_KAN_Weights".w2[399] * #v1[7] + "NeuroPLC_KAN_Weights".w2[400] * #v1[8] + "NeuroPLC_KAN_Weights".w2[401] * #v1[9] + "NeuroPLC_KAN_Weights".w2[402] * #v1[10] + "NeuroPLC_KAN_Weights".w2[403] * #v1[11] + "NeuroPLC_KAN_Weights".w2[404] * #v1[12] + "NeuroPLC_KAN_Weights".w2[405] * #v1[13] + "NeuroPLC_KAN_Weights".w2[406] * #v1[14] + "NeuroPLC_KAN_Weights".w2[407] * #v1[15] + "NeuroPLC_KAN_Weights".w2[408] * #v1[16] + "NeuroPLC_KAN_Weights".w2[409] * #v1[17] + "NeuroPLC_KAN_Weights".w2[410] * #v1[18] + "NeuroPLC_KAN_Weights".w2[411] * #v1[19] + "NeuroPLC_KAN_Weights".w2[412] * #v1[20] + "NeuroPLC_KAN_Weights".w2[413] * #v1[21] + "NeuroPLC_KAN_Weights".w2[414] * #v1[22] + "NeuroPLC_KAN_Weights".w2[415] * #v1[23] + "NeuroPLC_KAN_Weights".w2[416] * #v1[24] + "NeuroPLC_KAN_Weights".w2[417] * #v1[25] + "NeuroPLC_KAN_Weights".w2[418] * #v1[26] + "NeuroPLC_KAN_Weights".w2[419] * #v1[27];
          #v2[15] := "NeuroPLC_KAN_Weights".b3[15] + "NeuroPLC_KAN_Weights".w2[420] * #v1[0] + "NeuroPLC_KAN_Weights".w2[421] * #v1[1] + "NeuroPLC_KAN_Weights".w2[422] * #v1[2] + "NeuroPLC_KAN_Weights".w2[423] * #v1[3] + "NeuroPLC_KAN_Weights".w2[424] * #v1[4] + "NeuroPLC_KAN_Weights".w2[425] * #v1[5] + "NeuroPLC_KAN_Weights".w2[426] * #v1[6] + "NeuroPLC_KAN_Weights".w2[427] * #v1[7] + "NeuroPLC_KAN_Weights".w2[428] * #v1[8] + "NeuroPLC_KAN_Weights".w2[429] * #v1[9] + "NeuroPLC_KAN_Weights".w2[430] * #v1[10] + "NeuroPLC_KAN_Weights".w2[431] * #v1[11] + "NeuroPLC_KAN_Weights".w2[432] * #v1[12] + "NeuroPLC_KAN_Weights".w2[433] * #v1[13] + "NeuroPLC_KAN_Weights".w2[434] * #v1[14] + "NeuroPLC_KAN_Weights".w2[435] * #v1[15] + "NeuroPLC_KAN_Weights".w2[436] * #v1[16] + "NeuroPLC_KAN_Weights".w2[437] * #v1[17] + "NeuroPLC_KAN_Weights".w2[438] * #v1[18] + "NeuroPLC_KAN_Weights".w2[439] * #v1[19] + "NeuroPLC_KAN_Weights".w2[440] * #v1[20] + "NeuroPLC_KAN_Weights".w2[441] * #v1[21] + "NeuroPLC_KAN_Weights".w2[442] * #v1[22] + "NeuroPLC_KAN_Weights".w2[443] * #v1[23] + "NeuroPLC_KAN_Weights".w2[444] * #v1[24] + "NeuroPLC_KAN_Weights".w2[445] * #v1[25] + "NeuroPLC_KAN_Weights".w2[446] * #v1[26] + "NeuroPLC_KAN_Weights".w2[447] * #v1[27];

          // Add: l0_merge
          FOR #o := 0 TO 15 DO
              #sum := #v2[#o];  // base path
              FOR #i := 0 TO 27 DO
                  #idx := #o * 28 + #i;
                  #sum := #sum + #v3[#idx];  // spline path (1D)
              END_FOR;
              #v4[#o] := #sum;
          END_FOR;

          // StandardAct: silu
          FOR #i := 0 TO 15 DO
              // SiLU = x / (1 + exp(-x))
              #v5[#i] := #v4[#i] / (1.0 + EXP(-#v4[#i]));
          END_FOR;

          // BsplineLUT: l1_bspline (4x16, 15 pts)
          FOR #i := 0 TO 15 DO
              // Linear scan: find largest grid[j] <= input[i]
              #lo := 0;
              FOR #j := 1 TO 13 DO
                  IF #v4[#i] >= "NeuroPLC_KAN_Weights".g4[#j] THEN
                      #lo := #j;
                  END_IF;
              END_FOR;
              #hi := #lo + 1;
              #t_val := (#v4[#i] - "NeuroPLC_KAN_Weights".g4[#lo]) /
                        ("NeuroPLC_KAN_Weights".g4[#hi] - "NeuroPLC_KAN_Weights".g4[#lo] + 1.0E-10);
              FOR #o := 0 TO 3 DO
                  #base := (#o * 16 + #i) * 15;
                  #idx := #o * 16 + #i;
                  #v7[#idx] :=
                      "NeuroPLC_KAN_Weights".t5[#base + #lo] * (1.0 - #t_val) +
                      "NeuroPLC_KAN_Weights".t5[#base + #hi] * #t_val;
              END_FOR;
          END_FOR;

          // MatMul: l1_base
          #v6[0] := "NeuroPLC_KAN_Weights".b7[0] + "NeuroPLC_KAN_Weights".w6[0] * #v5[0] + "NeuroPLC_KAN_Weights".w6[1] * #v5[1] + "NeuroPLC_KAN_Weights".w6[2] * #v5[2] + "NeuroPLC_KAN_Weights".w6[3] * #v5[3] + "NeuroPLC_KAN_Weights".w6[4] * #v5[4] + "NeuroPLC_KAN_Weights".w6[5] * #v5[5] + "NeuroPLC_KAN_Weights".w6[6] * #v5[6] + "NeuroPLC_KAN_Weights".w6[7] * #v5[7] + "NeuroPLC_KAN_Weights".w6[8] * #v5[8] + "NeuroPLC_KAN_Weights".w6[9] * #v5[9] + "NeuroPLC_KAN_Weights".w6[10] * #v5[10] + "NeuroPLC_KAN_Weights".w6[11] * #v5[11] + "NeuroPLC_KAN_Weights".w6[12] * #v5[12] + "NeuroPLC_KAN_Weights".w6[13] * #v5[13] + "NeuroPLC_KAN_Weights".w6[14] * #v5[14] + "NeuroPLC_KAN_Weights".w6[15] * #v5[15];
          #v6[1] := "NeuroPLC_KAN_Weights".b7[1] + "NeuroPLC_KAN_Weights".w6[16] * #v5[0] + "NeuroPLC_KAN_Weights".w6[17] * #v5[1] + "NeuroPLC_KAN_Weights".w6[18] * #v5[2] + "NeuroPLC_KAN_Weights".w6[19] * #v5[3] + "NeuroPLC_KAN_Weights".w6[20] * #v5[4] + "NeuroPLC_KAN_Weights".w6[21] * #v5[5] + "NeuroPLC_KAN_Weights".w6[22] * #v5[6] + "NeuroPLC_KAN_Weights".w6[23] * #v5[7] + "NeuroPLC_KAN_Weights".w6[24] * #v5[8] + "NeuroPLC_KAN_Weights".w6[25] * #v5[9] + "NeuroPLC_KAN_Weights".w6[26] * #v5[10] + "NeuroPLC_KAN_Weights".w6[27] * #v5[11] + "NeuroPLC_KAN_Weights".w6[28] * #v5[12] + "NeuroPLC_KAN_Weights".w6[29] * #v5[13] + "NeuroPLC_KAN_Weights".w6[30] * #v5[14] + "NeuroPLC_KAN_Weights".w6[31] * #v5[15];
          #v6[2] := "NeuroPLC_KAN_Weights".b7[2] + "NeuroPLC_KAN_Weights".w6[32] * #v5[0] + "NeuroPLC_KAN_Weights".w6[33] * #v5[1] + "NeuroPLC_KAN_Weights".w6[34] * #v5[2] + "NeuroPLC_KAN_Weights".w6[35] * #v5[3] + "NeuroPLC_KAN_Weights".w6[36] * #v5[4] + "NeuroPLC_KAN_Weights".w6[37] * #v5[5] + "NeuroPLC_KAN_Weights".w6[38] * #v5[6] + "NeuroPLC_KAN_Weights".w6[39] * #v5[7] + "NeuroPLC_KAN_Weights".w6[40] * #v5[8] + "NeuroPLC_KAN_Weights".w6[41] * #v5[9] + "NeuroPLC_KAN_Weights".w6[42] * #v5[10] + "NeuroPLC_KAN_Weights".w6[43] * #v5[11] + "NeuroPLC_KAN_Weights".w6[44] * #v5[12] + "NeuroPLC_KAN_Weights".w6[45] * #v5[13] + "NeuroPLC_KAN_Weights".w6[46] * #v5[14] + "NeuroPLC_KAN_Weights".w6[47] * #v5[15];
          #v6[3] := "NeuroPLC_KAN_Weights".b7[3] + "NeuroPLC_KAN_Weights".w6[48] * #v5[0] + "NeuroPLC_KAN_Weights".w6[49] * #v5[1] + "NeuroPLC_KAN_Weights".w6[50] * #v5[2] + "NeuroPLC_KAN_Weights".w6[51] * #v5[3] + "NeuroPLC_KAN_Weights".w6[52] * #v5[4] + "NeuroPLC_KAN_Weights".w6[53] * #v5[5] + "NeuroPLC_KAN_Weights".w6[54] * #v5[6] + "NeuroPLC_KAN_Weights".w6[55] * #v5[7] + "NeuroPLC_KAN_Weights".w6[56] * #v5[8] + "NeuroPLC_KAN_Weights".w6[57] * #v5[9] + "NeuroPLC_KAN_Weights".w6[58] * #v5[10] + "NeuroPLC_KAN_Weights".w6[59] * #v5[11] + "NeuroPLC_KAN_Weights".w6[60] * #v5[12] + "NeuroPLC_KAN_Weights".w6[61] * #v5[13] + "NeuroPLC_KAN_Weights".w6[62] * #v5[14] + "NeuroPLC_KAN_Weights".w6[63] * #v5[15];

          // Add: l1_merge
          FOR #o := 0 TO 3 DO
              #sum := #v6[#o];  // base path
              FOR #i := 0 TO 15 DO
                  #idx := #o * 16 + #i;
                  #sum := #sum + #v7[#idx];  // spline path (1D)
              END_FOR;
              #v8[#o] := #sum;
          END_FOR;

          // Softmax
          #max_val := #v8[0];
          FOR #i := 1 TO 3 DO
              IF #v8[#i] > #max_val THEN
                  #max_val := #v8[#i];
              END_IF;
          END_FOR;
          #sum := 0.0;
          FOR #i := 0 TO 3 DO
              #v9[#i] := EXP(#v8[#i] - #max_val);
              #sum := #sum + #v9[#i];
          END_FOR;
          FOR #i := 0 TO 3 DO
              #v9[#i] := #v9[#i] / #sum;
          END_FOR;

          // Argmax
          #max_val := #v9[0];
          #fault_class := 0;
          FOR #i := 1 TO 3 DO
              IF #v9[#i] > #max_val THEN
                  #max_val := #v9[#i];
                  #fault_class := #i;
              END_IF;
          END_FOR;
          #confidence := #max_val;
END_FUNCTION_BLOCK

ORGANIZATION_BLOCK "Main"   // OB1, LAD, ProgramCycle
TITLE = "Main Program Sweep (Cycle)"
{ S7_Optimized_Access := 'TRUE' }
VERSION : 0.1
   VAR_INPUT
      Initial_Call : Bool;   // Initial call of this OB
      Remanence : Bool;   // =True, if remanent data are available
   END_VAR
BEGIN
END_ORGANIZATION_BLOCK